FUNCTION_BLOCK Q_NumericValue_PHYS_LREAL (* Command change numeric value — accepts NumericObjectPool_S struct and LREAL ( Part 6 - F.22 ) *)
  (* Standard: ISO 11783-6; Description: Copyright (c) 2026 Meisterschulen am Ostbahnhof This program and the accompanying materials are made available under the terms of the Eclipse Public License 2.0 which is available at https://www.eclipse.org/legal/epl-2.0/ SPDX-License-Identifier: EPL-2.0 *)
  (* Version 1.0, 2026-04-21, Franz Höpfinger, Meisterschulen am Ostbahnhof, initial API and implementation *)
  PACKAGE isobus::UT::Q;
  IMPORT eclipse4diac::core::TypeHash;
  IMPORT isobus::UT::Q::const::IDs::ID_NULL;
  IMPORT logiBUS::utils::conversion::phys::NumericObjectPool_S;
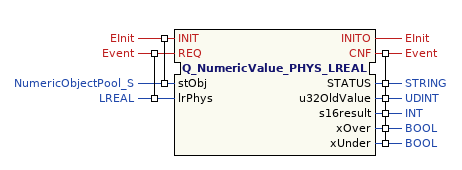
  EVENT_INPUT
    INIT : EInit WITH stObj; (* Service Initialization *)
    REQ WITH lrPhys; (* Service Request *)
  END_EVENT
  EVENT_OUTPUT
    INITO : EInit; (* Initialization Confirm *)
    CNF WITH STATUS, u32OldValue, s16result, xOver, xUnder; (* Confirmation of Requested Service *)
  END_EVENT
  VAR_INPUT
    stObj : logiBUS::utils::conversion::phys::NumericObjectPool_S := (u16ObjId := ID_NULL, r32Scale := 1.0, i32Offset := 0, u8Decimals := 0); (* Object pool properties (u16ObjId, scale, offset, decimals) *)
    lrPhys : LREAL; (* New raw value — use F_PHYS_LREAL_TO_RAW to convert from physical value *)
  END_VAR
  VAR_OUTPUT
    STATUS : STRING; (* Service Status *)
    u32OldValue : UDINT; (* Old raw value of ID *)
    s16result : INT; (* retval see Q_NumericValue *)
    xOver : BOOL; (* Physical value exceeds upper ISOBUS limit *)
    xUnder : BOOL; (* Physical value below lower ISOBUS limit *)
  END_VAR
  FBS
    Q_NumericValue : isobus::UT::Q::Q_NumericValue;
    F_PHYS_LREAL_TO_RAW : logiBUS::utils::conversion::phys::F_PHYS_LREAL_TO_RAW;
    F_MOVE : iec61131::selection::F_MOVE; {SET_ATTRIBUTE(DataType, logiBUS::utils::conversion::phys::NumericObjectPool_S)}
  END_FBS
  EVENT_CONNECTIONS
    Q_NumericValue.INITO TO INITO;
    Q_NumericValue.CNF TO CNF;
    F_PHYS_LREAL_TO_RAW.CNF TO Q_NumericValue.REQ;
    INIT TO F_MOVE.REQ;
    REQ TO F_PHYS_LREAL_TO_RAW.REQ;
    F_MOVE.CNF TO Q_NumericValue.INIT;
  END_CONNECTIONS
  DATA_CONNECTIONS
    Q_NumericValue.STATUS TO STATUS;
    Q_NumericValue.u32OldValue TO u32OldValue;
    Q_NumericValue.s16result TO s16result;
    stObj TO F_PHYS_LREAL_TO_RAW.stObj;
    F_PHYS_LREAL_TO_RAW. TO Q_NumericValue.u32NewValue;
    lrPhys TO F_PHYS_LREAL_TO_RAW.lrPhys;
    stObj TO F_MOVE.IN;
    F_MOVE.OUT.u16ObjId TO Q_NumericValue.u16ObjId;
    F_PHYS_LREAL_TO_RAW.xOver TO xOver;
    F_PHYS_LREAL_TO_RAW.xUnder TO xUnder;
  END_CONNECTIONS
END_FUNCTION_BLOCK
